FUNCTION_BLOCK FB_VFCModbus2 IMPLEMENTS I_VolumeFlowController
VAR_INPUT CONSTANT
	fbModbusMaster	:	POINTER TO FB_TVJModbusMaster;
	nUnitID			:	BYTE;
END_VAR
VAR_OUTPUT
END_VAR
VAR
	//Properties
	bError 			: 	BOOL := FALSE;
	fNominalVolFlow	: 	REAL := 8820;
	fVolFlowSet 	: 	REAL := 0;
	fVolFlowAct		: 	REAL;
	
	bFinish 		:	BOOL;
	
END_VAR

PROPERTY Error : BOOL
GET
Error := THIS^.bError;
END_GET
SET
THIS^.bError := Error;
END_SET
END_PROPERTY

PROPERTY NominalVolumeFlow : REAL
GET
NominalVolumeFlow := THIS^.fNominalVolFlow;
END_GET
SET
THIS^.fNominalVolFlow := NominalVolumeFlow;
END_SET
END_PROPERTY

METHOD Run : BOOL
//Write properties to master
fbModbusMaster^.NominalVolumeFlow := fNominalVolFlow;
fbModbusMaster^.VolumeFlowSetpoint := fVolFlowSet;
fbModbusMaster^.UnitID := nUnitID;

//Execute modbus master
bFinish := fbModbusMaster^.Run();

//Read properties from master
bError := fbModbusMaster^.Error;
IF bFinish THEN
	fVolFlowAct := fbModbusMaster^.VolumeFlowActual;
END_IF

Run := bFinish;
END_METHOD

PROPERTY UnitID : BYTE
GET
UnitID := THIS^.nUnitID;
END_GET
SET
THIS^.nUnitID := UnitID;
END_SET
END_PROPERTY

PROPERTY VolumeFlowActual : REAL
GET
VolumeFlowActual := THIS^.fVolFlowAct;
END_GET
SET
THIS^.fVolFlowAct := VolumeFlowActual;
END_SET
END_PROPERTY

PROPERTY VolumeFlowSetpoint : REAL
GET
VolumeFlowSetpoint := THIS^.fVolFlowSet;
END_GET
SET
THIS^.fVolFlowSet := VolumeFlowSetpoint;
END_SET
END_PROPERTY

END_FUNCTION_BLOCK

(* stored: Version 1.1.0.1, ProductVersion 3.1.4024.0
   POU FB_VFCModbus2: Id {7bb26802-ec16-4cae-86ee-6536cfe67ecc}, SpecialFunc None
   Property Error: Id {1e4d4fc0-1e4f-413d-9dda-bd74b12fddbe}
   Get Get: Id {c781e559-36b8-480d-b359-30ec89c68d51}
   Set Set: Id {fe1e28b0-7779-4aaa-b5cd-477382304475}
   Property NominalVolumeFlow: Id {22c2ccc8-abc0-4ab4-bbf3-11f46e572420}
   Get Get: Id {80e4a7d2-fa89-4683-91d1-735c93010f42}
   Set Set: Id {9e6dedcc-3c18-4bcd-924c-487c1b328cf1}
   Method Run: Id {edcc6de9-5878-481b-977b-59be4c6b2d3f}
   Property UnitID: Id {f74f62f6-22f1-4d66-bc95-6b3a6aeffe06}
   Get Get: Id {3263f6eb-a789-47df-957c-f0d6a3ed8912}
   Set Set: Id {040e9948-d15b-447c-ba31-3e136cd610f5}
   Property VolumeFlowActual: Id {9d30cb86-ad58-4bee-bf0f-49522bab7892}
   Get Get: Id {1760fb0e-19af-47be-8367-6ea31b0fb933}
   Set Set: Id {363d9a41-e0c9-42bf-8321-1ba45f6393d2}
   Property VolumeFlowSetpoint: Id {7b13ff72-b881-4065-97b0-46ae419b213c}
   Get Get: Id {3db50d7c-53fa-4e4f-b962-0217b3baee58}
   Set Set: Id {46124e2b-c604-4d67-960c-72d3bc0c1234} *)
